PROGRAM MAIN
VAR
	
	stWorkTime 				: ST_WorkTime;
	autoScadaLed			: Led;
	supplyScadaLed			: Led;
	statusScadaLabel		: Label;
	motorContactor 			: MotorContactor;
	motorTermFuse			: MotorTermFuse;
	autoScadaButton			: Button_NO;
	forwardScadaButton		: Button_NO;
	reverseScadaButton		: Button_NO;
	stateTaurusLed			: TaurusLed(forwardScadaButton, motorTermFuse);
	motorWorkTime 			: WorkCounter;
	
	

	
END_VAR



stateTaurusLed();
motorWorkTime();
motorWorkTime.CheckState(stateTaurusLed);

END_PROGRAM

(* stored: Version 1.1.0.1, ProductVersion 3.1.4024.12
   POU MAIN: Id {5ce869a2-8876-462e-9766-a690c22efe4d}, SpecialFunc None *)
